TYPE ST_INPUTS_ValveOnOFF:
STRUCT
	
	Mode:     	E_DeviceMode;
	Command:     E_DeviceState;

END_STRUCT
END_TYPE

(* stored: Version 1.1.0.1, ProductVersion 3.1.4024.12
   DUT ST_INPUTS_ValveOnOFF: Id {11da0b68-fcc2-4a88-b001-92e03af3eb78} *)
